SUBAPPLICATION AX_2_TO_3 (* UP/DOWN durchgereicht + gemeinsames ODER (z.B. Treiber-Enable) als drittes Signal - kein generischer ODER+SPLIT-Baustein, siehe AX_2_3 dafuer *)
  (* Standard: 61499-2; Description: Copyright (c) 2026 HR Agrartechnik GmbH This program and the accompanying materials are made available under the terms of the Eclipse Public License 2.0 which is available at https://www.eclipse.org/legal/epl-2.0/ SPDX-License-Identifier: EPL-2.0 *)
  (* Version 1.0, 2026-04-19, Franz Höpfinger, HR Agrartechnik GmbH *)
  PACKAGE MyLib::sys;
  (* Documentation:
  UP/DOWN-Passthrough plus gemeinsames ODER als drittes Signal
   Kein generischer ODER+SPLIT-Baustein wie AX_2_2/AX_2_3/ AX_3_2/AX_3_3, auch wenn der Name das nahelegt. Für einen Zweirichtungs-Aktor (z.B. Rechtslauf/Linkslauf eines Motors):
    - UP_IN und DOWN_IN werden je einzeln unverändert an UP_OUT bzw. DOWN_OUT durchgereicht (je ein eigener AX_SPLIT_2, damit beide Richtungen weiterhin getrennt an ihre jeweiligen physischen Ausgänge gehen).
   - Zusätzlich liefert OR_OUT das ODER aus UP_IN und DOWN_IN - "läuft der Aktor gerade in irgendeine Richtung" - z.B. um einen gemeinsamen Treiber/Enable-Ausgang (Low-Side-Treiber, Freigabe) zu schalten, der für beide Richtungen gebraucht wird.
    Reale Verwendung: Uebung_201b_AX…Uebung_205b_AX, dort speist ein Interlock (ILOCK_AX) UP_IN/DOWN_IN, und OR_OUT schaltet den gemeinsamen Treiber, während UP_OUT/DOWN_OUT die einzelnen Richtungsausgänge (Rechtslauf/Linkslauf) treiben.
   Für eine echte generische "N Quellen ODER-verknüpft auf M Ziele verteilt"-Konvertierung ohne Passthrough-Semantik stattdessen AX_2_3 verwenden. Werden UP/DOWN im Rest der Schaltung als gebündeltes A2X statt als zwei einzelne AX-Signale geführt, A2X_TO_A2X_AX verwenden (gleiches Prinzip, aber A2X-Ein-/Ausgang statt UP_IN/DOWN_IN und UP_OUT/DOWN_OUT).
  *)
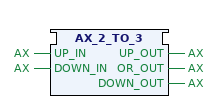
  SOCKETS
    UP_IN : adapter::types::unidirectional::AX;
    DOWN_IN : adapter::types::unidirectional::AX;
  END_SOCKETS
  PLUGS
    UP_OUT : adapter::types::unidirectional::AX;
    OR_OUT : adapter::types::unidirectional::AX;
    DOWN_OUT : adapter::types::unidirectional::AX;
  END_PLUGS
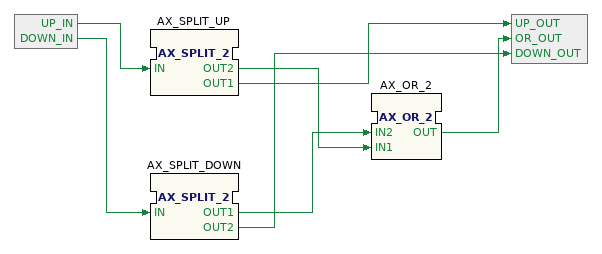
  FBS
    AX_SPLIT_DOWN : adapter::events::unidirectional::AX_SPLIT_2;
    AX_SPLIT_UP : adapter::events::unidirectional::AX_SPLIT_2;
    AX_OR_2 : adapter::booleanOperators::AX_OR_2;
  END_FBS
  ADAPTER_CONNECTIONS
    AX_SPLIT_DOWN.OUT1 TO AX_OR_2.IN2;
    AX_SPLIT_UP.OUT2 TO AX_OR_2.IN1;
    DOWN_IN TO AX_SPLIT_DOWN.IN;
    AX_SPLIT_DOWN.OUT2 TO DOWN_OUT;
    UP_IN TO AX_SPLIT_UP.IN;
    AX_SPLIT_UP.OUT1 TO UP_OUT;
    AX_OR_2.OUT TO OR_OUT;
  END_CONNECTIONS
END_SUBAPPLICATION
